FUNCTION_BLOCK XOR_4 (* FB to calculate bitwise boolean XOR (generic FB) *)
  (* Standard: 61131-3; Classification: standard bitwise boolean function; Description: Copyright (c) 2014 Profactor GmbH This program and the accompanying materials are made available under the terms of the Eclipse Public License 2.0 which is available at https://www.eclipse.org/legal/epl-2.0/ SPDX-License-Identifier: EPL-2.0 *)
  (* Version 1.0, 2014-10-11, Matthias Plasch, Profactor GmbH *)
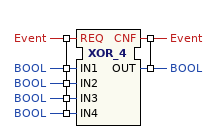
  EVENT_INPUT
    REQ WITH IN1, IN2, IN3, IN4; (* Normal Execution Request *)
  END_EVENT
  EVENT_OUTPUT
    CNF WITH OUT; (* Execution Confirmation *)
  END_EVENT
  VAR_INPUT
    IN1 : BOOL; (* XOR input 1 *)
    IN2 : BOOL; (* XOR input 2 *)
    IN3 : BOOL; (* XOR input 3 *)
    IN4 : BOOL; (* XOR input 4 *)
  END_VAR
  VAR_OUTPUT
    OUT : BOOL; (* XOR result *)
  END_VAR
END_FUNCTION_BLOCK
